// TIA Portal project "Batch_Automation_project" (V17)

(* hardware
DEVICE "S7-1200 station_1"  S7-1200 Station
   slot 0: "Rack_0"  S7-1200 Rack  Rack  V1.0
   slot 1: "PLC_1"  CPU 1215C DC/DC/DC  6ES7 215-1AG40-0XB0  V4.5
DEVICE "HMI_1"  TP700 Comfort
   slot 0: "HMI_1"  TP700 Comfort  6AV2 124-0GC01-0AX0  17.0.0.0
   slot 1: "HMI_RT_1"  TP700 Comfort  6AV2 124-0GC01-0AX0  17.0.0.0
   slot 5: "HMI_1.IE_CP_1"  PROFINET Interface  17.0.0.0
      slot 1: "PROFINET Interface_1"  PROFINET Interface
         slot 1: "Port_1"  Port
         slot 2: "Port_2"  Port
   slot 7: "HMI_1.MPI/DP_CP_1"  MPI/DP Interface  17.0.0.0
*)

// ===== PLC "PLC_1"  CPU 1215C DC/DC/DC =====

VAR_GLOBAL   // PLC tag table "Default tag table"
   "Start_Batch" AT %I0.0 : Bool;   // Start bacth command
   "Stop_Batch" AT %I0.1 : Bool;   // Stoop batch command
   "Level_Low" AT %I0.2 : Bool;   // Tank low level sensor
   "Level_High" AT %I0.3 : Bool;   // Tank high level sensor
   "Drain_Empty" AT %I0.4 : Bool;   // Tank empty after drain
   "Agitator_FB" AT %I0.5 : Bool;   // Agitator running feedback
   "Fault_Reset" AT %I0.6 : Bool;   // Fault reset button
   "Recipe_Select" AT %I0.7 : Bool;   // 0=recipe1,1=recipe2
   "Value_A" AT %Q0.0 : Bool;   // Ingredient A inlet value
   "Value_B" AT %Q0.1 : Bool;   // Ingredient B inlet value
   "Agitator" AT %Q0.2 : Bool;   // Mixing agitator motor
   "Heater" AT %Q0.3 : Bool;   // Tank heater
   "Drain_Value" AT %Q0.4 : Bool;   // Product drain value
   "Batch_Complete" AT %Q0.5 : Bool;   // Batch done indicator
   "Fault_Light" AT %Q0.6 : Bool;   // Fault alarm ligt
   "Temp_raw" AT %ID64 : Real;   // Temperature 4-20mA
   "Heater_Output" AT %QD68 : Real;   // heater power 0-100%
END_VAR

TYPE "Recipe_UDT"
   STRUCT
      Fill_Level : Real;   // Target Fill%
      Mix_Time : Time;   // Mixing Duration
      Heat_Temp : Real;   // Target temperatur C
      Hold_time : Time;   // Hold at temperature
      Recipe_Name : String;   // Recipe Description
   END_STRUCT;
END_TYPE

DATA_BLOCK "Recipe1_DB"   // DB1
{ S7_Optimized_Access := 'TRUE' }
VERSION : 0.1
   VAR
      Recipe : "Recipe_UDT";
   END_VAR
BEGIN
   Recipe.Fill_Level := 80.0;
   Recipe.Mix_Time := T#5M;
   Recipe.Heat_Temp := 60.0;
   Recipe.Hold_time := T#2M;
   Recipe.Recipe_Name := 'Standard Mix';
END_DATA_BLOCK

DATA_BLOCK "Recipe2_DB"   // DB2
{ S7_Optimized_Access := 'TRUE' }
VERSION : 0.1
   VAR
      Recipe2 : "Recipe_UDT";
   END_VAR
BEGIN
   Recipe2.Fill_Level := 90.0;
   Recipe2.Mix_Time := T#8M;
   Recipe2.Heat_Temp := 75.0;
   Recipe2.Hold_time := T#3M;
   Recipe2.Recipe_Name := 'Concentrated Mix';
END_DATA_BLOCK

DATA_BLOCK "Batch_DB"   // DB3
{ S7_Optimized_Access := 'TRUE' }
VERSION : 0.1
   VAR
      Batch_State : Int;   // Current State 0-7
      Batch_Running : Bool;   // Batch active flag
      Batch_Complete : Bool;   // Batch finished flag
      Fault_Active : Bool;   // Any fault present
      Fault_Code : Int;   // Which fault(0=none)
      Recipe_Number : Int;   // Active recipe(1 r 2)
      Current_Temp : Real;   // Scaled temperature
      Fill_Percent : Real;   // current fill level
      Batch_Count : Int;   // total batched completed
      Phase_Name : String;   // current phase name
      Heater_Cv : Real;   // PID Output %
      Fill_Target : Real := 80.0;
      Mix_Duration : Time := T#5M;
      Heat_Target : Real := 60.0;
      Hold_Duration : Time := T#2M;
      Temp_Wire_Break : Bool;
      Temp_Overflow : Bool;
      Fill_Waiting : Bool;
      Fill_Active : Bool;
      Fill_Complete : Bool;
      Mix_Waiting : Bool;
      Mix_Active : Bool;
      Mix_Complete : Bool;
      Heat_Waiting : Bool;
      Heat_Active : Bool;
      Heat_Complete : Bool;
      Drain_Waiting : Bool;
      Drain_Active : Bool;
      Drain_Complete : Bool;
   END_VAR
BEGIN
END_DATA_BLOCK

DATA_BLOCK "Fill_DB"   // DB4
{ S7_Optimized_Access := 'TRUE' }
VERSION : 0.1
// stored: InstanceOfName Fill_Phase
"Fill_Phase"
BEGIN
END_DATA_BLOCK

DATA_BLOCK "Mix_DB"   // DB5
{ S7_Optimized_Access := 'TRUE' }
VERSION : 0.1
// stored: InstanceOfName Mix_Phase
"Mix_Phase"
BEGIN
END_DATA_BLOCK

DATA_BLOCK "Heat_DB"   // DB6
{ S7_Optimized_Access := 'TRUE' }
VERSION : 0.1
// stored: InstanceOfName Heat_Phase
"Heat_Phase"
BEGIN
END_DATA_BLOCK

DATA_BLOCK "Drain_DB"   // DB7
{ S7_Optimized_Access := 'TRUE' }
VERSION : 0.1
// stored: InstanceOfName Drain_Phase
"Drain_Phase"
BEGIN
END_DATA_BLOCK

DATA_BLOCK "Alarm_DB"   // DB8
{ S7_Optimized_Access := 'TRUE' }
VERSION : 0.1
   VAR
      Alarm_Word : Word;
   END_VAR
BEGIN
END_DATA_BLOCK

FUNCTION_BLOCK "Fill_Phase"   // FB1, SCL
{ S7_Optimized_Access := 'TRUE' }
VERSION : 0.1
   VAR_INPUT
      Execute : Bool;
      Target_Level : Real;
      Level_High : Bool;
      Abort : Bool;
   END_VAR
   VAR_OUTPUT
      Running : Bool;
      Done : Bool;
      Fault : Bool;
      Value_A_cmd : Bool;
      Value_B_cmd : Bool;
   END_VAR
   VAR
      Phase_State : Int;
      Fill_TImer : TON_TIME;
   END_VAR
BEGIN
   // FILL PHASE FB
   // States: 0=Idle 1=Filling 2=Done 3=Fault

   //Abort from any state
   IF #Abort THEN
       #Phase_State := 3;
   END_IF;

   CASE #Phase_State OF
       0: //IDLE - waiting for execute
           #Running := FALSE;
           #Done := FALSE;
           #Value_A_cmd := FALSE;
           #Value_B_cmd := FALSE;

           IF #Execute THEN
               #Phase_State := 1;
           END_IF;

       1: //Filling - open valves
           #Running := TRUE;
           #Done := FALSE;
           #Value_A_cmd := TRUE;
           #Value_B_cmd := TRUE;

           //waitfor high level sensor
           IF #Level_High THEN
               #Value_A_cmd := FALSE;
               #Value_B_cmd := FALSE;
               #Phase_State := 2;
           END_IF;

       2://done
           #Running := FALSE;
           #Done := TRUE;
           #Value_A_cmd := FALSE;
           #Value_B_cmd := FALSE;

           IF NOT #Execute THEN
               #Phase_State := 0;
           END_IF;

       3: //fault
           #Running := FALSE;
           #Done := FALSE;
           #Fault := TRUE;
           #Value_A_cmd := FALSE;
           #Value_B_cmd := FALSE;

       ELSE
           #Phase_State := 0;
   END_CASE;
END_FUNCTION_BLOCK

FUNCTION_BLOCK "Mix_Phase"   // FB2, SCL
{ S7_Optimized_Access := 'TRUE' }
VERSION : 0.1
   VAR_INPUT
      Execute : Bool;
      Target_Level : Real;
      Level_High : Bool;
      Abort : Bool;
      Mix_Duration : Time;
   END_VAR
   VAR_OUTPUT
      Running : Bool;
      Done : Bool;
      Fault : Bool;
      Agitator_CMD : Bool;
   END_VAR
   VAR
      Phase_State : Int;
      Mix_Timer : TON_TIME;
   END_VAR
BEGIN
   // MIX PHASE FB
   // States: 0=Idle 1=Mixing 2=Done 3=Fault

   //Abort from any state
   IF #Abort THEN
       #Phase_State := 3;
   END_IF;

   CASE #Phase_State OF
       0: //IDLE - waiting for execute
           #Running := FALSE;
           #Done := FALSE;
           #Agitator_CMD := FALSE;
           #Mix_Timer(IN := FALSE, PT:=#Mix_Duration);

           IF #Execute THEN
               #Phase_State := 1;
           END_IF;

       1: //MIXING
           #Running := TRUE;
           #Agitator_CMD := FALSE;
           #Mix_Timer(IN := TRUE,
                      PT := #Mix_Duration);

           //waitfor high level sensor
           IF #Mix_Timer.Q THEN
               #Phase_State := 2;
           END_IF;

       2://done
           #Running := FALSE;
           #Done := TRUE;
           #Agitator_CMD := FALSE;

           IF NOT #Execute THEN
               #Phase_State := 0;
           END_IF;

       3: //fault
           #Running := FALSE;
           #Done := FALSE;
           #Fault := TRUE;
           #Agitator_CMD := FALSE;

       ELSE
           #Phase_State := 0;
   END_CASE;
END_FUNCTION_BLOCK

FUNCTION_BLOCK "Heat_Phase"   // FB3, SCL
{ S7_Optimized_Access := 'TRUE' }
VERSION : 0.1
   VAR_INPUT
      Execute : Bool;
      Target_Temp : Real;
      Current_Temp : Real;
      Abort : Bool;
      Hold_Duration : Time;
      Current_Mode : Int;
   END_VAR
   VAR_OUTPUT
      Running : Bool;
      Done : Bool;
      Fault : Bool;
      Heater_CMD : Bool;
      Heater_Power : Real;
   END_VAR
   VAR
      Phase_State : Int;
      Hold_TImer : TON_TIME;
      Temp_PID : PID_Compact;
   END_VAR
BEGIN
   // HEAT PHASE FB
   // States: 0=Idle 1=Heating 2=Holding 3=Done 4=Fault

   //Abort from any state
   IF #Abort THEN
       #Phase_State := 4;
   END_IF;

   CASE #Phase_State OF
       0: //IDLE - waiting for execute
           #Running := FALSE;
           #Done := FALSE;
           #Heater_CMD := FALSE;
           #Heater_Power := 0.0;
           #Hold_TImer(IN := FALSE,
                       PT := #Hold_Duration);

           IF #Execute THEN
               #Phase_State := 1;
           END_IF;

       1: //HEATING - PID controls heater
           #Running := TRUE;
           #Done := FALSE;
           #Temp_PID(Setpoint:=#Target_Temp, Input:=#Current_Temp, Output=>#Heater_Power, Mode := #Current_Mode);

           #Heater_CMD := #Heater_Power > 5.0;

           //waitfor high level sensor
           IF #Current_Temp >= (#Target_Temp - 2.0) THEN
               #Phase_State := 2;
           END_IF;

       2://HOLDING
           #Running := TRUE;
           #Done := FALSE;
           #Temp_PID(Setpoint:=#Target_Temp, Input:=#Current_Temp, Output=>#Heater_Power, Mode:=#Current_Mode);

           #Heater_CMD := #Heater_Power > 5.0;

           #Hold_TImer(IN := TRUE,
                       PT := #Hold_Duration);

           IF #Hold_TImer.Q THEN
               #Phase_State := 3;
           END_IF;

       3: //Done
           #Running := FALSE;
           #Done := TRUE;
           #Heater_CMD := FALSE;
           #Heater_Power := 0.0;
           #Hold_TImer(IN := FALSE,
                       PT := #Hold_Duration);

           IF NOT #Execute THEN
               #Phase_State := 0;
           END_IF;

       4: //fault
           #Running := FALSE;
           #Done := FALSE;
           #Fault := TRUE;
           #Heater_CMD := FALSE;
           #Heater_Power := 0.0;

   END_CASE;
END_FUNCTION_BLOCK

FUNCTION_BLOCK "Drain_Phase"   // FB4, SCL
{ S7_Optimized_Access := 'TRUE' }
VERSION : 0.1
   VAR_INPUT
      Execute : Bool;
      Tank_Empty : Bool;
      Abort : Bool;
   END_VAR
   VAR_OUTPUT
      Running : Bool;
      Done : Bool;
      Fault : Bool;
      Drain_Valu_CMD : Bool;
   END_VAR
   VAR
      Phase_State : Int;
      Drain_Timeout : TON_TIME;
   END_VAR
BEGIN
   // DRAIN PHASE FB
   // States: 0=Idle 1=Draining 2=Done 3=Fault

   //Abort from any state
   IF #Abort THEN
       #Phase_State := 3;
   END_IF;

   CASE #Phase_State OF
       0: //IDLE - waiting for execute
           #Running := FALSE;
           #Done := FALSE;
           #Drain_Valu_CMD := FALSE;
           #Drain_Timeout(IN := FALSE,
                          PT := T#5S);

           IF #Execute THEN
               #Phase_State := 1;
           END_IF;

       1: //Draining
           #Running := TRUE;
           #Drain_Valu_CMD := TRUE;
           #Drain_Timeout(IN := FALSE,
                          PT := T#5S);

           //waitfor high level sensor
           IF #Tank_Empty THEN
               #Phase_State := 2;
           ELSIF #Drain_Timeout.Q THEN
               #Phase_State := 3;
           END_IF;

       2://Done
           #Running := FALSE;
           #Done := TRUE;
           #Drain_Valu_CMD := FALSE;

           IF NOT #Execute THEN
               #Phase_State := 0;
           END_IF;

      3: //fault
           #Running := FALSE;
           #Done := FALSE;
           #Fault := TRUE;
           #Drain_Valu_CMD := FALSE;

   END_CASE;
END_FUNCTION_BLOCK

FUNCTION "Recipe_Manager" : Void   // FC1, SCL
{ S7_Optimized_Access := 'TRUE' }
VERSION : 0.1
   VAR_INPUT
      Recipe_Select : Bool;
   END_VAR
   VAR_OUTPUT
      Fill_Level : Real;
      Mix_Time : Time;
      Heat_Temp : Real;
      Hold_Time : Time;
   END_VAR
BEGIN
   //RECIPE MANAGER
   //Recipe_Select False = Recipe 1
   //Recipe_Select True = Recipe 2

   IF NOT #Recipe_Select THEN
       // Recipe 1 - Standard Mix
       #Fill_Level := "Recipe1_DB".Recipe.Fill_Level;
       #Mix_Time := "Recipe1_DB".Recipe.Mix_Time;
       #Heat_Temp := "Recipe1_DB".Recipe.Heat_Temp;
       #Hold_Time := "Recipe1_DB".Recipe.Hold_time;
   ELSE
       // Recipe 2 - Concentrated Mix
       #Fill_Level := "Recipe2_DB".Recipe2.Fill_Level;
       #Mix_Time := "Recipe2_DB".Recipe2.Mix_Time;
       #Heat_Temp := "Recipe2_DB".Recipe2.Heat_Temp;
       #Hold_Time := "Recipe2_DB".Recipe2.Hold_time;
   END_IF;
END_FUNCTION

FUNCTION "Analog_Scaling" : Void   // FC2, SCL
{ S7_Optimized_Access := 'TRUE' }
VERSION : 0.1
   VAR_INPUT
      Raw_Value : Int;
      Eng_Min : Real;
      Eng_Max : Real;
      Raw_Min : Int;
      Raw_Max : Int;
   END_VAR
   VAR_OUTPUT
      Eng_Value : Real;
      Wire_Break : Bool;
      Overflow : Bool;
   END_VAR
BEGIN
   // Analog Scaling

   //Wire break detection
   IF #Raw_Value < 1000 THEN
       #Wire_Break := TRUE;
       #Eng_Value := 0.0;
       RETURN;
   END_IF;

   //Overflow detection
   IF #Raw_Value > 28000 THEN
       #Overflow := TRUE;
       #Eng_Value := #Eng_Max;
       RETURN;
   END_IF;

   //Normal Scaling
   #Wire_Break := FALSE;
   #Overflow := FALSE;

   #Eng_Value := (INT_TO_REAL(#Raw_Value - #Raw_Min) *
                   (#Eng_Max - #Eng_Min)) /
                   INT_TO_REAL(#Raw_Max - #Raw_Min) +
                   #Eng_Min;
END_FUNCTION

FUNCTION "Alarm_Handler" : Void   // FC3, SCL
{ S7_Optimized_Access := 'TRUE' }
VERSION : 0.1
BEGIN
END_FUNCTION

ORGANIZATION_BLOCK "Main"   // OB1, SCL, ProgramCycle
TITLE = "Main Program Sweep (Cycle)"
{ S7_Optimized_Access := 'TRUE' }
VERSION : 0.1
   VAR_INPUT
      Initial_Call : Bool;   // Initial call of this OB
      Remanence : Bool;   // =True, if remanent data are available
   END_VAR
BEGIN
   //=====================================
   //BATCH AUTOMATION - MASTER SEQUENCE
   //PROJECT 3 - S88 BATCH CONTROL
   //=====================================

   //Step 1 - Get Recipe Paramters
   "Recipe_Manager"(Recipe_Select:="Recipe_Select",
                    Fill_Level=>"Batch_DB".Fill_Target,
                    Mix_Time=>"Batch_DB".Mix_Duration,
                    Heat_Temp=>"Batch_DB".Heat_Target,
                    Hold_Time=>"Batch_DB".Hold_Duration);

   //Step 2 - Scale Temperature
   "Analog_Scaling"(Raw_Value:="Temp_raw",
                    Eng_Min:=0.0,
                    Eng_Max:=150.0,
                    Raw_Min:=0,
                    Raw_Max:=27648,
                    Eng_Value=>"Batch_DB".Current_Temp,
                    Wire_Break=>"Batch_DB".Temp_Wire_Break,
                    Overflow=>"Batch_DB".Temp_Overflow);

   //Step 3 - Master Batch State Machine
   //States: 0-IDLE 1=FILL 2=MIX 3=HEAT 4=DRAIN 5=DONE

   //Emergency abort from any state
   IF "Stop_Batch" THEN
       "Batch_DB".Batch_State := 0;
       "Batch_DB".Batch_Running := FALSE;
   END_IF;

   CASE "Batch_DB".Batch_State OF
       0: //IDLE - Waiting for start
           "Batch_DB".Batch_Running := FALSE;
           "Batch_DB".Batch_Complete := FALSE;
           "Batch_DB".Phase_Name := 'IDLE';

           IF "Start_Batch" AND NOT "Batch_DB".Fault_Active THEN
               "Batch_DB".Batch_State := 1;
               "Batch_DB".Batch_Running := TRUE;
           END_IF;

       1: //FILL PHASE
           "Batch_DB".Phase_Name := 'FILLING';

           "Fill_DB"(Execute := TRUE,
                     Target_Level := "Batch_DB".Fill_Target,
                     Level_High := "Level_High",
                     Abort := "Stop_Batch");

           "Value_A" := "Fill_DB".Value_A_cmd;
           "Value_B" := "Fill_DB".Value_B_cmd;

           IF "Fill_DB".Done THEN
               "Fill_DB"(Execute := FALSE,
                         Target_Level := 0.0,
                         Level_High := FALSE,
                         Abort := FALSE);
               "Batch_DB".Batch_State := 2;
           ELSIF "Fill_DB".Fault THEN
               "Batch_DB".Fault_Active := TRUE;
               "Batch_DB".Fault_Code := 1;
               "Batch_DB".Batch_State := 0;
           END_IF;

       2: //MIX PHASE
           "Batch_DB".Phase_Name := 'MIXING';

           "Mix_DB"(Execute := TRUE,
                    Mix_Duration := "Batch_DB".Mix_Duration,
                     Abort := "Stop_Batch");

            "Agitator" := "Mix_DB".Agitator_CMD;

           IF "Mix_DB".Done THEN
               "Mix_DB"(Execute := FALSE,
                        Mix_Duration := T#0S,
                        Abort := FALSE);
               "Batch_DB".Batch_State := 3;
           ELSIF "Mix_DB".Fault THEN
               "Batch_DB".Fault_Active := TRUE;
               "Batch_DB".Fault_Code := 2;
               "Batch_DB".Batch_State := 0;
           END_IF;

       3: //HEAT PHASE
           "Batch_DB".Phase_Name := 'HEATING';

           "Heat_DB"(Execute := TRUE,
                     Target_Temp := "Batch_DB".Heat_Target,
                     Current_Temp := "Batch_DB".Current_Temp,
                     Hold_Duration := "Batch_DB".Hold_Duration,
                    Abort := "Stop_Batch");

          "Heater" := "Heat_DB".Heater_CMD;
          "Batch_DB".Heater_Cv := "Heat_DB".Heater_Power;

          IF "Heat_DB".Done THEN
              "Heat_DB"(Execute := FALSE,
                        Target_Temp := 0.0,
                        Current_Temp := 0.0,
                        Hold_Duration := T#0S,
                        Abort := FALSE);
              "Batch_DB".Batch_State := 4;
          ELSIF "Heat_DB".Fault THEN
              "Batch_DB".Fault_Active := TRUE;
              "Batch_DB".Fault_Code := 3;
              "Batch_DB".Batch_State := 0;
          END_IF;

      4: //DRAIN PHASE
          "Batch_DB".Phase_Name := 'DRAINING';

          "Drain_DB"(Execute := TRUE,
                     Tank_Empty := "Drain_Empty",
                     Abort := "Stop_Batch");

         "Drain_Value" := "Drain_DB".Drain_Valu_CMD;

          IF "Drain_DB".Done THEN
              "Drain_DB"(Execute := FALSE,
                         Tank_Empty := FALSE,
                        Abort := FALSE);
             "Batch_DB".Batch_State := 5;
             "Batch_DB".Batch_Count := "Batch_DB".Batch_Count + 1;
          ELSIF "Drain_DB".Fault THEN
              "Batch_DB".Fault_Active := TRUE;
              "Batch_DB".Fault_Code := 4;
              "Batch_DB".Batch_State := 0;
          END_IF;

      5: // DONE
          "Batch_DB".Phase_Name := 'COMPLETE';
          "Batch_DB".Batch_Running := FALSE;
          "Batch_DB".Batch_Complete := TRUE;
          "Batch_Complete" := TRUE;

          //Auto reset after 5 seconds
          IF NOT "Start_Batch" THEN
              "Batch_DB".Batch_State := 0;
              "Batch_DB".Batch_Complete := FALSE;
              "Batch_Complete" := FALSE;
          END_IF;

   END_CASE;

   //Fill Status
   "Batch_DB".Fill_Waiting := NOT "Fill_DB".Running AND NOT "Fill_DB".Done;
   "Batch_DB".Fill_Active := "Fill_DB".Running;
   "Batch_DB".Fill_Complete := "Fill_DB".Done;

   //Mix Status
   "Batch_DB".Mix_Waiting := NOT "Mix_DB".Running AND NOT "Mix_DB".Done;
   "Batch_DB".Mix_Active := "Mix_DB".Running;
   "Batch_DB".Mix_Complete := "Mix_DB".Done;

   //Heat Status
   "Batch_DB".Heat_Waiting := NOT "Heat_DB".Running AND NOT "Heat_DB".Done;
   "Batch_DB".Heat_Active := "Heat_DB".Running;
   "Batch_DB".Heat_Complete := "Heat_DB".Done;

   //Drain Status
   "Batch_DB".Drain_Waiting := NOT "Drain_DB".Running AND NOT "Drain_DB".Done;
   "Batch_DB".Drain_Active := "Drain_DB".Running;
   "Batch_DB".Drain_Complete := "Drain_DB".Done;

   //Step 4 : Fault Handling
   IF "Batch_DB".Fault_Active THEN
       "Fault_Light" := TRUE;

       //Reset fault with button
       IF "Fault_Reset" THEN
           "Batch_DB".Fault_Active := FALSE;
           "Batch_DB".Fault_Code := 0;
           "Fault_Light" := FALSE;
       END_IF;
   END_IF;

   //Step 5 - Write Master Analog Output
   "Heater_Output" := REAL_TO_INT("Batch_DB".Heater_Cv / 100.0 * 27648.0);
END_ORGANIZATION_BLOCK

(* ===== HMI "HMI_RT_1" =====
system functions are stored by id; their names below are inferred from use
connection "HMI_Connection_1": ETHERNET, S7_1200_OMS

HMI tags "Default tag table"
   "Start_Batch" : Bool = PLC Start_Batch AT %I0.0, 1 s
   "Stop_Batch" : Bool = PLC Stop_Batch AT %I0.1, 1 s
   "Fault_Reset" : Bool = PLC Fault_Reset AT %I0.6, 1 s
   "Batch_Complete" : Bool = PLC Batch_Complete AT %Q0.5, 1 s
   "Batch_State" : Int = PLC Batch_DB.Batch_State AT %DB1.DBX0.0, 1 s
   "Batch_Running" : Bool = PLC Batch_DB.Batch_Running AT %DB1.DBW0, 1 s
   "Phase_Name" : String[254] = PLC Batch_DB.Phase_Name AT %DB1.DBX0.0, 1 s
   "Recipe_Number" : Int = PLC Batch_DB.Recipe_Number AT %DB1.DBX0.0, 1 s
   "Current_Temp" : Real = PLC Batch_DB.Current_Temp AT %DB1.DBW0, 1 s
   "Fault_active" : Bool = PLC Batch_DB.Fault_Active AT %DB1.DBD0, 1 s
   "Batch_Count" : Int = PLC Batch_DB.Batch_Count AT %DB1.DBX0.0, 1 s
   "Heater_Cv" : Real = PLC Batch_DB.Heater_Cv AT %DB1.DBW0, 1 s
   "Heat_Target" : Real = PLC Batch_DB.Heat_Target AT %DB1.DBD0, 1 s
   "Fill_Running" : Bool = PLC Fill_DB.Running AT %DB1.DBD0, 1 s
   "Fault_Code" : Int = PLC Batch_DB.Fault_Code AT %DB1.DBW0, 1 s
   "Fill_Done" : Bool = PLC Fill_DB.Done AT %DB1.DBX0.0, 1 s
   "Mix_Running" : Bool = PLC Mix_DB.Running AT %DB1.DBX0.0, 1 s
   "Mix_DOne" : Bool = PLC Mix_DB.Done AT %DB1.DBX0.0, 1 s
   "Heat_Running" : Bool = PLC Heat_DB.Running AT %DB1.DBX0.0, 1 s
   "Heat_Done" : Bool = PLC Heat_DB.Done AT %DB1.DBX0.0, 1 s
   "Drain_Running" : Bool = PLC Drain_DB.Running AT %DB1.DBX0.0, 1 s
   "Drain_Done" : Bool = PLC Drain_DB.Done AT %DB1.DBX0.0, 1 s
   "Reipe_Select" : Bool = PLC Recipe_Select AT %I0.7, 1 s
   "Alarm_Word" : Word = PLC Alarm_DB.Alarm_Word AT %DB1.DBX0.0, 1 s
   "Fill_wait" : Bool = PLC Batch_DB.Fill_Waiting AT %DB1.DBW0, 1 s
   "Fill_Active" : Bool = PLC Batch_DB.Fill_Active AT %DB1.DBX0.0, 1 s
   "Fill_Complete" : Bool = PLC Batch_DB.Fill_Complete AT %DB1.DBX0.0, 1 s
   "Mix_Wait" : Bool = PLC Batch_DB.Mix_Waiting AT %DB1.DBX0.0, 1 s
   "Mix_Active" : Bool = PLC Batch_DB.Mix_Active AT %DB1.DBX0.0, 1 s
   "Mix_Complete" : Bool = PLC Batch_DB.Mix_Complete AT %DB1.DBX0.0, 1 s
   "Heat_Mix" : Bool = PLC Batch_DB.Heat_Waiting AT %DB1.DBX0.0, 1 s
   "Heat_Active" : Bool = PLC Batch_DB.Heat_Active AT %DB1.DBX0.0, 1 s
   "Heat_Complete" : Bool = PLC Batch_DB.Heat_Complete AT %DB1.DBX0.0, 1 s
   "Drain_Mix" : Bool = PLC Batch_DB.Drain_Waiting AT %DB1.DBX0.0, 1 s
   "Drain_Active" : Bool = PLC Batch_DB.Drain_Active AT %DB1.DBX0.0, 1 s
   "Drain_Complete" : Bool = PLC Batch_DB.Drain_Complete AT %DB1.DBX0.0, 1 s

discrete alarms
   1: '', class Errors, trigger "Alarm_Word" bit 0
   2: '', class Errors, trigger "Heater_Cv" bit 0
   3: '', class Errors, trigger "Alarm_Word" bit 2
   4: '', class Errors, trigger "Alarm_Word" bit 3
   5: '', class Errors, trigger "Alarm_Word" bit 1

Template "Template_1" 800x420
   Button "Exit" at 720,360 size 78x58; TextOff 'Exit'; PictureOff "ExitRuntime_TP700_Comfort_TR"; PictureOn "ExitRuntime_TP700_Comfort_TR"
      on Release: StopRuntime(0)
   Button "Template_Button" at 640,360 size 78x58; TextOff 'Text'
   Button "Template_Button_1" at 560,360 size 78x58; TextOff 'Text'
   Button "Template_Button_2" at 480,360 size 78x58; TextOff 'Text'
   Button "Template_Button_3" at 400,360 size 78x58; TextOff 'Text'
   Button "Template_Button_4" at 321,360 size 78x58; TextOff 'Text'
   Button "Template_Button_5" at 241,360 size 78x58; TextOff 'Text'
   Button "Template_Button_6" at 161,360 size 78x58; TextOff 'Text'
   Button "Alarms" at 81,360 size 78x58; TextOff 'Alarms'; PictureOff "AlarmDisplay_TP700_Comfort_TR"; PictureOn "AlarmDisplay_TP700_Comfort_TR"
      on Release: function_ef3f5d25("Alarm window_Unacknowledged", -1)
   Button "Start screen" at 1,360 size 78x58; TextOff 'Start screen'; PictureOff "NavigateHome_TP700_Comfort_TR"; PictureOn "NavigateHome_TP700_Comfort_TR"
      on Release: ActivateScreen("Root screen", 0)

screen "Alarm_Screen" 800x420
   AlarmView "Alarm view_1" at 13,44 size 739x316
   Button "Button_4" at 689,372 size 63x45; TextOff 'Home'
      on Activate: ActivateScreen("Root screen", 0)
   TextField "Text field_1" at 283,14 size 151x23; Text 'Alarm Screen'

screen "Trends/History" 800x420
   TrendView "Trend view_1" at 38,42 size 697x317
   Button "Button_4" at 693,364 size 63x45; TextOff 'Home'
      on Activate: ActivateScreen("Root screen", 0)
   TextField "Text field_1" at 300,7 size 173x23; Text 'Trend Screen'

screen "Root screen" 800x420, template "Template_1"
   on GenerateScreen: SetTag("Start_Batch", 1)
   Button "Button_1" at 93,15 size 80x33; TextOff 'START'
      on Press: SetBit("Start_Batch")
   Button "Button_2" at 197,15 size 80x33; TextOn 'STOP'; TextOff 'STOP'
      on Press: SetBit("Stop_Batch")
   Button "Button_3" at 301,15 size 80x33; TextOn 'RESET'; TextOff 'RESET'
      on Press: SetBit("Fault_Reset")
   IOField "I/O field_1" at 271,67 size 150x34; FormatPattern ????????????????????
      ProcessValue <- "Phase_Name"
   TextField "Text field_1" at 93,71 size 168x26; Text 'CURRENT PHASE:'
   TextField "Text field_2" at 93,111 size 168x26; Text 'STATE:'
   IOField "I/O field_2" at 166,109 size 61x32; FormatPattern s99
      ProcessValue <- "Batch_State"
   TextField "Text field_3" at 277,111 size 209x26; Text 'BATCHES COMPLETED:'
   IOField "I/O field_3" at 494,109 size 76x32; FormatPattern s999
      ProcessValue <- "Batch_Count"
   TextField "Text field_4" at 117,171 size 69x30; Text 'FILL ✅'
      Visibility <- "Fill_Complete"
   TextField "Text field_6" at 277,159 size 209x26; Text 'TEMPERATURE:'
   IOField "I/O field_4" at 494,157 size 76x32; FormatPattern 999.9
      ProcessValue <- "Current_Temp"
   TextField "Text field_5" at 277,207 size 209x26; Text 'TARGET:'
   IOField "I/O field_5" at 494,205 size 76x32; FormatPattern 999.9
      ProcessValue <- "Heat_Target"
   Bar "Bar_1" at 441,15 size 201x77; MinimumValue 0; MaximumValue 100
      ProcessValue <- "Heater_Cv"
   IOField "I/O field_6" at 654,45 size 76x32; FormatPattern 999
      ProcessValue <- "Heater_Cv"
   TextField "Text field_7" at 423,257 size 248x23; Text '⚠ FAULT ACTIVE — CODE:'
      Visibility <- "Fault_active"
   Button "Button_4" at 649,369 size 63x45; TextOff 'Alarms'
      on Activate: ActivateScreen("Alarm_Screen", 0)
   Button "Button_5" at 569,369 size 63x45; TextOff 'Recipe'
      on Activate: ActivateScreen("Recipe_selection", 0)
   Button "Button_6" at 489,369 size 63x45; TextOff 'Trends'
      on Activate: ActivateScreen("Trends/History", 0)
   IOField "I/O field_7" at 685,251 size 49x32; FormatPattern 9
      ProcessValue <- "Fault_Code"
   TextField "Text field_8" at 117,171 size 69x30; Text 'FILL'
      Visibility <- "Fill_wait"
   TextField "Text field_9" at 117,171 size 69x30; Text 'FILL'
      Visibility <- "Fill_Active"
   TextField "Text field_10" at 118,237 size 69x30; Text 'MIX'
      Visibility <- "Mix_Active"
   TextField "Text field_11" at 117,297 size 76x30; Text 'DRAIN'
      Visibility <- "Drain_Active"
   TextField "Text field_12" at 118,237 size 69x30; Text 'MIX ✅'
      Visibility <- "Mix_Complete"
   TextField "Text field_13" at 117,297 size 82x30; Text 'DRAIN ✅'
      Visibility <- "Drain_Complete"
   TextField "Text field_14" at 118,237 size 69x30; Text 'MIX'
      Visibility <- "Mix_Wait"
   TextField "Text field_15" at 117,297 size 82x30; Text 'DRAIN'
      Visibility <- "Drain_Mix"

screen "Recipe_selection" 800x420
   TextField "Text field_12" at 229,20 size 231x26; Text 'Recipe Selection'
   TextField "Text field_7" at 127,73 size 274x23; Text 'Recipe 1 - STANDARD MIX'
   TextField "Text field_2" at 127,107 size 256x23; Text 'Fill Level : 80%'
   TextField "Text field_3" at 127,139 size 256x23; Text 'Mix Time : 5 Minutes'
   TextField "Text field_4" at 127,171 size 256x26; Text 'Heat Temp : 60 C'
   TextField "Text field_5" at 127,203 size 256x23; Text 'Hold Time : 2 Minutes'
   Button "Button_1" at 127,235 size 167x35; TextOff 'Select Recipe 1'
      on Click: ResetBit("Reipe_Select")
      Appearance <- "Reipe_Select"
   TextField "Text field_1" at 439,72 size 279x23; Text 'Recipe 2 - CONCENTRATED'
   TextField "Text field_8" at 439,107 size 267x23; Text 'Fill Level : 90%'
   TextField "Text field_9" at 439,139 size 267x23; Text 'Mix Time : 8 Minutes'
   TextField "Text field_10" at 439,171 size 267x23; Text 'Heat Temp : 75 C'
   TextField "Text field_11" at 439,203 size 267x23; Text 'Hold Time : 3 Minutes'
   Button "Button_2" at 439,235 size 172x34; TextOff 'Select Recipe 2'
      on Click: SetBit("Reipe_Select")
      Appearance <- "Reipe_Select"
   IOField "I/O field_1" at 329,300 size 60x31; FormatPattern 9
      ProcessValue <- "Recipe_Number"
   TextField "Text field_6" at 177,301 size 136x23; Text 'Active Recipe:'
   Button "Button_4" at 693,348 size 63x45; TextOff 'Home'
      on Activate: ActivateScreen("Root screen", 0)
*)